(* Schneider Machine Expert - Basic project A2, file version 1.8.0.0 *)
(* ProjectInformations: Name=New project *)

HARDWARE
  Cpu 0: TM221CE16R
  EthernetConfiguration: NetworkName=M221, IpAllocationMode=FixedAddress, IpAddress=192.168.162.202, SubnetMask=255.255.255.0
  SerialLineConfiguration: Baud=Baud19200, Parity=ParityEven, DataBits=DataBits8, StopBits=StopBits1, PhysicalMedium=PhysicalMediumRs485, TransmissionMode=TransmissionModeModbusRtu, SlaveId=1, Addressing=SlaveAddressing
  MastTask: UsePeriodScanMode=false, PeriodScan=100
  FastTask: Period=255
  CpuBehavior: StartingMode=StartAsPreviousState, AutoSaveRamOnEeprom=true, WatchdogPeriod=250

SYMBOLS  (address, symbol, comment, settings)
  %TM0        [Preset=1, Base=OneSecond]
  %TM1        [Preset=1, Base=OneSecond]
  %TM2        [Preset=1, Base=OneSecond]
  %TM3        [Preset=1, Base=OneSecond]

POU start/stop
  (* SectionNumber=1 *)

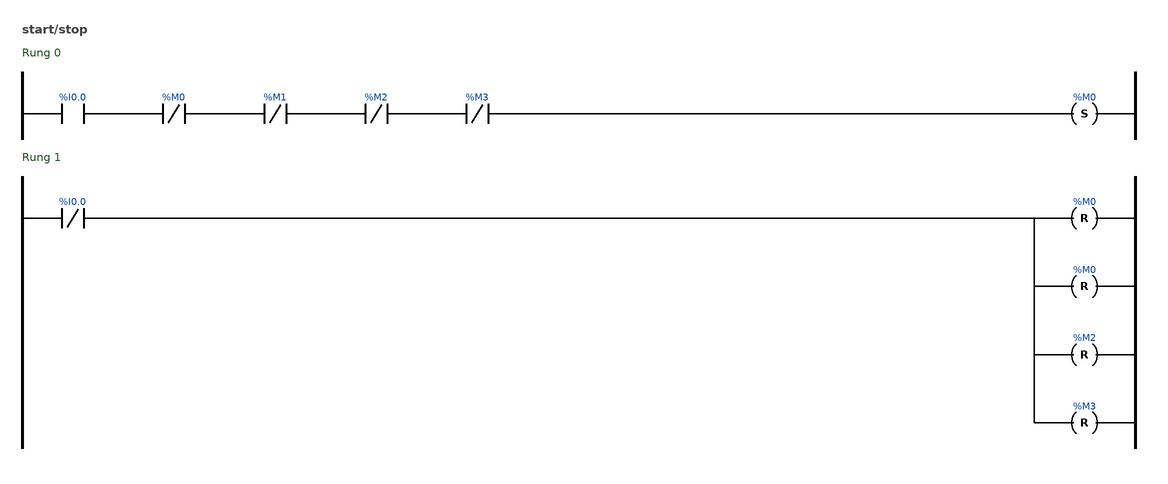

// Rung 0
  LD %I0.0
  ANDN %M0
  ANDN %M1
  ANDN %M2
  ANDN %M3
  S %M0
  // as ST:
  //   IF %I0.0 AND NOT %M0 AND NOT %M1 AND NOT %M2 AND NOT %M3 THEN %M0 := TRUE; END_IF;

// Rung 1
  LDN %I0.0
  R %M0
  R %M0
  R %M2
  R %M3
  // as ST:
  //   IF NOT %I0.0 THEN %M0 := FALSE; END_IF;
  //   IF NOT %I0.0 THEN %M0 := FALSE; END_IF;
  //   IF NOT %I0.0 THEN %M2 := FALSE; END_IF;
  //   IF NOT %I0.0 THEN %M3 := FALSE; END_IF;

POU timer
  (* SectionNumber=2 *)

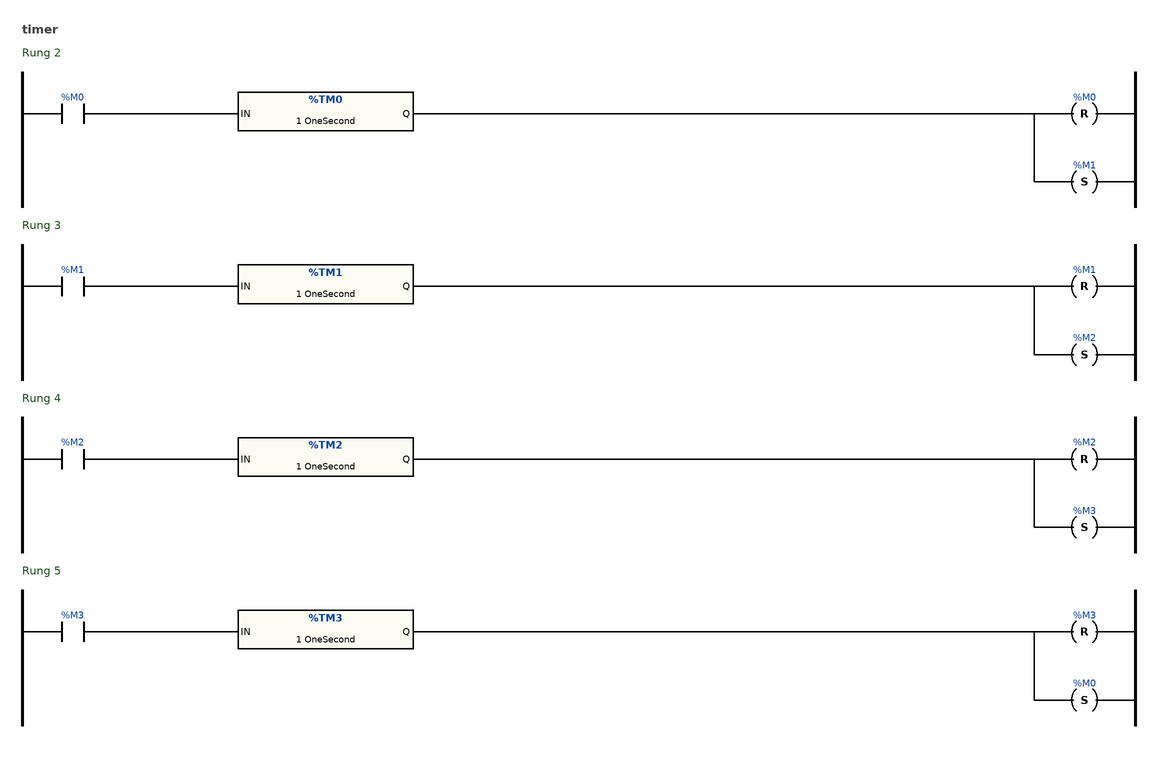

// Rung 2
  BLK %TM0
  LD %M0
  IN
  OUT_BLK
  LD Q
  R %M0
  S %M1
  END_BLK
  // as ST:
  //   %TM0(IN := %M0);
  //   IF %TM0.Q THEN %M0 := FALSE; END_IF;
  //   IF %TM0.Q THEN %M1 := TRUE; END_IF;

// Rung 3
  BLK %TM1
  LD %M1
  IN
  OUT_BLK
  LD Q
  R %M1
  S %M2
  END_BLK
  // as ST:
  //   %TM1(IN := %M1);
  //   IF %TM1.Q THEN %M1 := FALSE; END_IF;
  //   IF %TM1.Q THEN %M2 := TRUE; END_IF;

// Rung 4
  BLK %TM2
  LD %M2
  IN
  OUT_BLK
  LD Q
  R %M2
  S %M3
  END_BLK
  // as ST:
  //   %TM2(IN := %M2);
  //   IF %TM2.Q THEN %M2 := FALSE; END_IF;
  //   IF %TM2.Q THEN %M3 := TRUE; END_IF;

// Rung 5
  BLK %TM3
  LD %M3
  IN
  OUT_BLK
  LD Q
  R %M3
  S %M0
  END_BLK
  // as ST:
  //   %TM3(IN := %M3);
  //   IF %TM3.Q THEN %M3 := FALSE; END_IF;
  //   IF %TM3.Q THEN %M0 := TRUE; END_IF;

POU DecodeOutput
  (* SectionNumber=3 *)

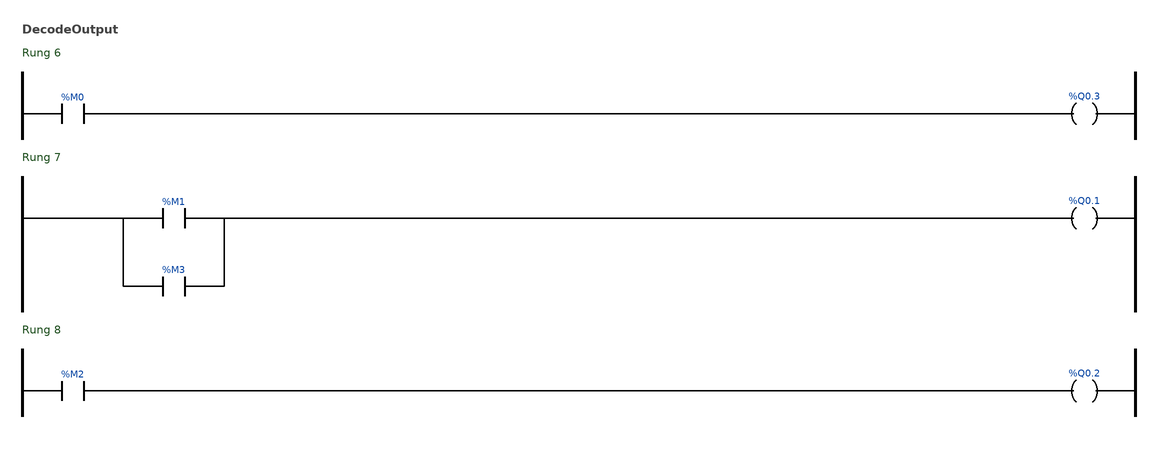

// Rung 6
  LD %M0
  ST %Q0.3
  // as ST:
  //   %Q0.3 := %M0;

// Rung 7
  LD %M1
  OR %M3
  ST %Q0.1
  // as ST:
  //   %Q0.1 := %M1 OR %M3;

// Rung 8
  LD %M2
  ST %Q0.2
  // as ST:
  //   %Q0.2 := %M2;
